(* PLC project mtcs_m3, Institute of Astronomy OntoManager 0.0.1 *)
(* stored: creationDateTime 2024-08-13T08:58:49.312185, modificationDateTime 2024-08-13T08:58:49.312185 *)

TYPE M3PositionIDs : (UNKNOWN := 0, CASSEGRAIN := 1, NASMYTH_A := 2, NASMYTH_B := 3, NASMYTH_C := 4, NASMYTH_D := 5, OTHER_0 := 6, OTHER_1 := 7, OTHER_2 := 8, OTHER_3 := 9, OTHER_4 := 10);
END_TYPE

TYPE M3GotoProcedureStates : (IDLE := 0, ABORTED := 1, PREPARE_PROCESS := 2, GOING_TO_POSITION := 3, IMPROVING_POSITION := 4, ERROR := 5, RESETTING := 6, ABORTING := 7);
END_TYPE

TYPE M3RotateProcedureStates : (IDLE := 0, ABORTED := 1, PREPARE_PROCESS := 2, DECOUPLING_AXES := 3, ENABLING_AXES := 4, UNDOING_OFFSET := 5, COUPLING_AXES := 6, BOTH_GOING_TO_TARGET_PLUS_OFFSET := 7, DECOUPLING_AXES_AGAIN := 8, MOVING_ABL_TO_FINAL_POSITION := 9, DISABLING_ABL := 10, MOVING_POS_TO_FINAL_POSITION := 11, IMPROVING_POSITION := 12, DISABLING_POS := 13, ERROR := 14, RESETTING := 15, ABORTING := 16);
END_TYPE

TYPE M3TranslateProcedureStates : (IDLE := 0, ABORTED := 1, PREPARE_PROCESS := 2, ENABLING_AXIS := 3, MOVING := 4, IMPROVING_POSITION := 5, DISABLING_AXIS := 6, ERROR := 7, RESETTING := 8, ABORTING := 9);
END_TYPE

TYPE M3TranslationHomingProcedureStates : (IDLE := 0, ABORTED := 1, PREPARE_PROCESS := 2, ENABLING_AXIS := 3, MOVE_TO_LIMIT_SWITCH := 4, WAIT_FOR_LIMIT_SWITCH := 5, STOP := 6, APPLY_HOMING_SETTINGS := 7, MOVE_TO_MECH_STOP := 8, WAIT_FOR_MECH_STOP := 9, SET_ZERO_POSITION := 10, DISABLE_AXIS := 11, RESETTING := 12, ERROR := 13, ABORTING := 14);
END_TYPE

TYPE M3CalibrateRotationProcedureStates : (IDLE := 0, ABORTED := 1, PREPARE_PROCESS := 2, DECOUPLING_AXES := 3, ENABLING_AXES := 4, COUPLING_AXES := 5, GOING_TO_START_POSITION := 6, DECOUPLING_AXES_AGAIN := 7, START_MOVING := 8, WAIT_UNTIL_MOVING_STABLE := 9, WAIT_UNTIL_RANGE_PASSED := 10, HALT := 11, GO_TO_CLUTCH_ZERO_TORQUE := 12, DISABLING_AXES := 13, WAIT_UNTIL_STANDSTILL := 14, SYNC_AXES := 15, ERROR := 16, RESETTING := 17, ABORTING := 18);
END_TYPE

TYPE M3TargetStates : (NO_TARGET_GIVEN := 0, KNOWN_POSITION := 1, NEW_POSITION := 2);
END_TYPE

TYPE M3Parts : STRUCT
  rotation : M3Rotation;  (* Rotation mechanism *)
  translation : M3Translation;  (* Translation mechanism *)
  io : M3IO;  (* I/O modules *)
  gotoProcedure : M3GotoProcedure;  (* The goto procedure *)
  configManager : ConfigManager;  (* The config manager (to load/save/activate configuration data) *)
END_STRUCT;
END_TYPE

TYPE M3RotationParts : STRUCT
  positioningAxis : AngularAxis;  (* Positioning axis: SSI encoder + Faulhaber drive *)
  antiBacklashAxis : AngularAxis;  (* Anti-backlash Axis: Faulhaber drive + hall sensors *)
  positioningDrive : FaulhaberDrive;  (* Positioning drive *)
  antiBacklashDrive : FaulhaberDrive;  (* Anti-backlash drive *)
  positioningHallAxis : AngularAxis;  (* Only hall sensors *)
  gotoProcedure : M3RotationGotoProcedure;  (* The goto procedure *)
  calibrateProcedure : M3RotationCalibrateProcedure;  (* The calibration procedure *)
END_STRUCT;
END_TYPE

TYPE M3TranslationParts : STRUCT
  motorAxis : LinearAxis;  (* Motor axis *)
  motorDrive : FaulhaberDrive;  (* Motor drive *)
  gotoProcedure : M3TranslationGotoProcedure;  (* The goto procedure *)
  homingProcedure : M3TranslationHomingProcedure;  (* The homing procedure *)
END_STRUCT;
END_TYPE

TYPE M3IOParts : STRUCT
  canOpenBus : CANopenBus;  (* CANopen bus *)
  coupler : EtherCatDevice;  (* Coupler *)
  slot1 : EtherCatDevice;  (* Slot 1 *)
  slot2 : EtherCatDevice;  (* Slot 2 *)
  slot3 : EtherCatDevice;  (* Slot 3 *)
  slot4 : EtherCatDevice;  (* Slot 4 *)
END_STRUCT;
END_TYPE

TYPE M3Processes : STRUCT
  initialize : Process;  (* Start initializing *)
  lock : Process;  (* Lock the system *)
  unlock : Process;  (* Unlock the system *)
  reset : Process;  (* Reset any errors *)
  changeOperatingState : ChangeOperatingStateProcess;  (* Change the operating state (e.g. AUTO, MANUAL, ...) *)
  gotoKnownPosition : M3GotoKnownPosition;  (* Go to the known position with the given name (only in AUTO mode!) *)
  gotoNewPosition : M3GotoNewPosition;  (* Go to the new position with the given settings (only in AUTO mode!) *)
  abort : Process;  (* Abort the goto procedure *)
END_STRUCT;
END_TYPE

TYPE M3RotationProcesses : STRUCT
  goto : M3RotationGoto;  (* Start moving the rotation stage to the given position *)
  abort : Process;  (* Abort any running procedures *)
  reset : Process;  (* Reset any errors *)
  calibrate : Process;  (* Start calibrating the rotation stage *)
END_STRUCT;
END_TYPE

TYPE M3TranslationProcesses : STRUCT
  goto : M3TranslationGoto;  (* Start moving the translation stage to the given position *)
  reset : Process;  (* Reset any errors *)
  abort : Process;  (* Abort any running procedures *)
  startHoming : Process;  (* Start the homing procedure *)
END_STRUCT;
END_TYPE

TYPE M3RotationTargetStatuses : STRUCT
  targetStatus : M3TargetStatus;
END_STRUCT;
END_TYPE

TYPE M3TranslationTargetStatuses : STRUCT
  targetStatus : M3TargetStatus;
END_STRUCT;
END_TYPE

TYPE M3Statuses : STRUCT
  initializationStatus : InitializationStatus;
  apertureStatus : ApertureStatus;
  healthStatus : HealthStatus;
  busyStatus : BusyStatus;
  operatingStatus : OperatingStatus;
END_STRUCT;
END_TYPE

TYPE M3GotoProcedureStatuses : STRUCT
  busyStatus : BusyStatus;  (* Is the M3GotoProcedure in a busy state? *)
  healthStatus : HealthStatus;  (* Is the M3GotoProcedure in a healthy state? *)
END_STRUCT;
END_TYPE

TYPE M3RotationStatuses : STRUCT
  healthStatus : HealthStatus;
  busyStatus : BusyStatus;
END_STRUCT;
END_TYPE

TYPE M3RotationGotoProcedureStatuses : STRUCT
  busyStatus : BusyStatus;  (* Is the M3RotationGotoProcedure in a busy state? *)
  healthStatus : HealthStatus;  (* Is the M3RotationGotoProcedure in a healthy state? *)
END_STRUCT;
END_TYPE

TYPE M3RotationCalibrateProcedureStatuses : STRUCT
  busyStatus : BusyStatus;  (* Is the M3RotationCalibrateProcedure in a busy state? *)
  healthStatus : HealthStatus;  (* Is the M3RotationCalibrateProcedure in a healthy state? *)
END_STRUCT;
END_TYPE

TYPE M3TranslationStatuses : STRUCT
  healthStatus : HealthStatus;
  busyStatus : BusyStatus;
END_STRUCT;
END_TYPE

TYPE M3TranslationGotoProcedureStatuses : STRUCT
  busyStatus : BusyStatus;  (* Is the M3GotoProcedure in a busy state? *)
  healthStatus : HealthStatus;  (* Is the M3GotoProcedure in a healthy state? *)
END_STRUCT;
END_TYPE

TYPE M3TranslationHomingProcedureStatuses : STRUCT
  busyStatus : BusyStatus;  (* Is the M3GotoProcedure in a busy state? *)
  healthStatus : HealthStatus;  (* Is the M3GotoProcedure in a healthy state? *)
END_STRUCT;
END_TYPE

TYPE M3IOStatuses : STRUCT
  healthStatus : HealthStatus;  (* Is the I/O in a healthy state? *)
END_STRUCT;
END_TYPE

TYPE M3PositionConfig : STRUCT
  name : STRING;  (* The name of the M3 position *)
  rotationPosition : LREAL;  (* The position of the rotation stage in degrees *)
  rotationOffset : LREAL;  (* The offset between the positions of the two motors of the rotation stage in degrees *)
  translationPosition : LREAL;  (* The position of the translation stage in millimeters *)
  doRotation : BOOL;  (* Do a rotation for this position (TRUE) or not (FALSE) *)
  doTranslation : BOOL;  (* Do a translation for this position (TRUE) or not (FALSE) *)
END_STRUCT;
END_TYPE

TYPE M3KnownPositionsConfig : STRUCT
  cassegrain : M3PositionConfig;  (* Cassegrain *)
  nasmythA : M3PositionConfig;  (* Nasmyth A *)
  nasmythB : M3PositionConfig;  (* Nasmyth B *)
  nasmythC : M3PositionConfig;  (* Nasmyth C *)
  nasmythD : M3PositionConfig;  (* Nasmyth D *)
  other0 : M3PositionConfig;  (* Freely choosable position 0 *)
  other1 : M3PositionConfig;  (* Freely choosable position 1 *)
  other2 : M3PositionConfig;  (* Freely choosable position 2 *)
  other3 : M3PositionConfig;  (* Freely choosable position 3 *)
  other4 : M3PositionConfig;  (* Freely choosable position 4 *)
END_STRUCT;
END_TYPE

TYPE M3RotationConfig : STRUCT
  standstillTolerance : LREAL;  (* The tolerance for which the axis appears to be standing still, in degrees/sec *)
  motorToMirrorRatio : LREAL;  (* The motor-to-mirror transmission ratio *)
  encoderToMirrorRatio : LREAL;  (* The encoder-to-mirror transmission ratio *)
  positioningDrive : FaulhaberDriveConfig;  (* The config of the positioning faulhaber drive *)
  antiBacklashDrive : FaulhaberDriveConfig;  (* The config of the anti-backlash faulhaber drive *)
  negativeSoftLimit : LREAL;  (* Negative soft limit, in degrees *)
  positiveSoftLimit : LREAL;  (* Negative soft limit, in degrees *)
  maxPositionError : LREAL;  (* Maximum position error, in degrees *)
  maxOffsetError : LREAL;  (* Maximum position error, in degrees *)
  gotoOffsetVelocity : LREAL;  (* Velocity to move from/to the offset position, in degrees/sec on the MOTOR reduction exit shaft reference system *)
  gotoTargetVelocity : LREAL;  (* Velocity to move to the target, in degrees/sec on the MIRROR reference system *)
  gotoImprovingPositionTime : LREAL;  (* Time while the Goto procedure may improve the position, in seconds *)
  calibrateStartPosition : LREAL;  (* Mirror position (in degrees) to start the calibration from *)
  calibrateMoveToZeroTorqueVelocity : LREAL;  (* Velocity to move to the zero-torque position, in degrees/sec on the MIRROR reference system *)
  calibrateVelocity : LREAL;  (* Velocity during which the current is being measured, in degrees/sec on the MIRROR reference system *)
  calibrateRange : LREAL;  (* Position range where the current is being measured, in degrees on the MOTOR reference system *)
  calibrateOffset : LREAL;  (* Degrees between zero-torque position and minimum-torque position, on the MOTOR reference system *)
END_STRUCT;
END_TYPE

TYPE M3TranslationConfig : STRUCT
  homingContinuousCurrentLimit : UINT;  (* The continuous current limit for the translation stage motor in milliAmps, during homing *)
  homingPeakCurrentLimit : UINT;  (* The peak current limit for the translation stage motor in milliAmps, during homing *)
  homingSearchLimitSwitchVelocity : LREAL;  (* The velocity of the motor shaft during homing, in mm/sec *)
  homingToHardwareStopVelocity : LREAL;  (* The velocity of the motor shaft during homing, in mm/sec *)
  standstillTolerance : LREAL;  (* The tolerance for which the axis appears to be standing still, in mm/sec *)
  motorDrive : FaulhaberDriveConfig;  (* The config of the faulhaber drive *)
  negativeSoftLimit : LREAL;  (* Negative soft limit, in millimeters *)
  positiveSoftLimit : LREAL;  (* Negative soft limit, in millimeters *)
  maxPositionError : LREAL;  (* Maximum position error, in millimeters *)
  drawCassegrainLimit : LREAL;  (* Below this limit (in millimeters) the mirror will be drawn flipped away *)
  drawNasmythLimit : LREAL;  (* Above this limit (in millimeters) the mirror will be drawn frontal *)
  gotoImprovingPositionTime : LREAL;  (* Time while the Goto procedure may improve the position, in seconds *)
  gotoVelocity : LREAL;  (* Velocity to go to a new position, in degrees/second *)
END_STRUCT;
END_TYPE

TYPE M3Config : STRUCT
  knownPositions : M3KnownPositionsConfig;  (* All known M3 positions *)
  rotation : M3RotationConfig;  (* The settings of the rotation stage *)
  translation : M3TranslationConfig;  (* The settings of the translation stage *)
  moveAfterInitialization : BOOL;  (* Move the mirror to a known position after initialization *)
  moveAfterInitializationPosition : STRING;  (* Move the mirror to this position after initialization *)
END_STRUCT;
END_TYPE

TYPE M3GotoKnownPositionArgs : STRUCT
  name : STRING;  (* Name of the position (must be configured in M3Config.knownPositions!) *)
END_STRUCT;
END_TYPE

TYPE M3GotoNewPositionArgs : STRUCT
  rotationPosition : LREAL;  (* Position of the rotation stage, in degrees *)
  rotationOffset : LREAL;  (* Offset between the motors of the rotation stage, in degrees *)
  translationPosition : LREAL;  (* Position of the rotation stage, in millimeters *)
  doRotation : BOOL;  (* Do a rotation for this position (TRUE) or not (FALSE) *)
  doTranslation : BOOL;  (* Do a translation for this position (TRUE) or not (FALSE) *)
END_STRUCT;
END_TYPE

TYPE M3RotationGotoArgs : STRUCT
  position : LREAL;  (* Position setpoint of the rotation stage, in degrees *)
  offset : LREAL;  (* Offset setpoint between the motors of the rotation stage, in degrees *)
END_STRUCT;
END_TYPE

TYPE M3TranslationGotoArgs : STRUCT
  position : LREAL;  (* Position setpoint of the translation stage, in millimeters *)
END_STRUCT;
END_TYPE

FUNCTION_BLOCK M3TargetStatus
  VAR_INPUT
    superState : BOOL := TRUE;  (* Super state (TRUE if the super state is active, or if there is no super state) *)
    state : M3TargetStates;  (* Enum! *)
  END_VAR
  VAR_OUTPUT
    {attribute 'OPC.UA.DA' := '1'}
    {attribute 'OPC.UA.DA.Access' := '1'}
    noTargetGiven : BOOL;  (* No target given *)
    {attribute 'OPC.UA.DA' := '1'}
    {attribute 'OPC.UA.DA.Access' := '1'}
    knownPosition : BOOL;  (* Known position *)
    {attribute 'OPC.UA.DA' := '1'}
    {attribute 'OPC.UA.DA.Access' := '1'}
    newPosition : BOOL;  (* Undefined *)
  END_VAR

            noTargetGiven := (state = M3TargetStates.NO_TARGET_GIVEN) AND superState;
knownPosition := (state = M3TargetStates.KNOWN_POSITION) AND superState;
newPosition := (state = M3TargetStates.NEW_POSITION) AND superState;

          
END_FUNCTION_BLOCK

FUNCTION_BLOCK SM_M3RotationTarget
  VAR_INPUT
    {attribute 'OPC.UA.DA' := '0'}
    isTargetGiven : BOOL;  (* TRUE if a target is given *)
    {attribute 'OPC.UA.DA' := '0'}
    newPositionDegrees : LREAL;  (* New target position in degrees *)
    {attribute 'OPC.UA.DA' := '0'}
    newOffsetDegrees : LREAL;  (* New target offset in degrees *)
  END_VAR
  VAR_OUTPUT
    {attribute 'OPC.UA.DA' := '1'}
    {attribute 'OPC.UA.DA.Access' := '1'}
    actualStatus : STRING;  (* Current status description *)
    previousStatus : STRING;  (* Previous status description *)
    {attribute 'OPC.UA.DA' := '1'}
    {attribute 'OPC.UA.DA.Access' := '1'}
    name : STRING;  (* Name of the target (only in case the position and offset match an entry in the config!) *)
    {attribute 'OPC.UA.DA' := '1'}
    {attribute 'OPC.UA.DA.Access' := '1'}
    position : AngularPosition;  (* Target position for M3 rotation (only in case statuses.targetStatus.noTargetGiven is FALSE) *)
    {attribute 'OPC.UA.DA' := '1'}
    {attribute 'OPC.UA.DA.Access' := '1'}
    offset : AngularPosition;  (* Target offset for M3 rotation (only in case statuses.targetStatus.noTargetGiven is FALSE) *)
    statuses : M3RotationTargetStatuses;  (* Statuses of the state machine *)
  END_VAR
  VAR_IN_OUT
    {attribute 'OPC.UA.DA' := '0'}
    knownPositions : M3KnownPositionsConfig;  (* The known positions *)
  END_VAR

            position( newDegreesValue := newPositionDegrees );
offset( newDegreesValue := newOffsetDegrees );
statuses.targetStatus();

          

{attribute 'TcRpcEnable' := '1'}
METHOD _log : BOOL
  VAR_INPUT
    name : STRING;  (* Name of this function block instance *)
  END_VAR
  VAR_IN_OUT
    buffer : LogBuffer;  (* Buffer to write all logging to *)
  END_VAR
  VAR
    subBuffer : LogBuffer;  (* Temporary buffer to write logging by parts (sub-statemachines) to *)
  END_VAR
                  LOGGER(
    name := name,
    actualStatus := THIS^.actualStatus,
    previousStatus := THIS^.previousStatus,
    buffer := buffer,
    subBuffer := subBuffer);

                
END_METHOD
END_FUNCTION_BLOCK

FUNCTION_BLOCK SM_M3TranslationTarget
  VAR_INPUT
    {attribute 'OPC.UA.DA' := '0'}
    isTargetGiven : BOOL := FALSE;  (* TRUE if a target is given *)
    {attribute 'OPC.UA.DA' := '0'}
    newPositionMillimeters : LREAL;  (* New target position in millimeters *)
  END_VAR
  VAR_OUTPUT
    {attribute 'OPC.UA.DA' := '1'}
    {attribute 'OPC.UA.DA.Access' := '1'}
    actualStatus : STRING;  (* Current status description *)
    previousStatus : STRING;  (* Previous status description *)
    {attribute 'OPC.UA.DA' := '1'}
    {attribute 'OPC.UA.DA.Access' := '1'}
    name : STRING;  (* Name of the target (only in case the position matches an entry in the config!) *)
    {attribute 'OPC.UA.DA' := '1'}
    {attribute 'OPC.UA.DA.Access' := '1'}
    position : LinearPosition;  (* Target position for M3 translation (only in case statuses.targetStatus.noTargetGiven is FALSE) *)
    statuses : M3TranslationTargetStatuses;  (* Statuses of the state machine *)
  END_VAR
  VAR_IN_OUT
    {attribute 'OPC.UA.DA' := '0'}
    knownPositions : M3KnownPositionsConfig;  (* The known positions *)
  END_VAR

            position( newMillimetersValue := newPositionMillimeters );
statuses.targetStatus();

          

{attribute 'TcRpcEnable' := '1'}
METHOD _log : BOOL
  VAR_INPUT
    name : STRING;  (* Name of this function block instance *)
  END_VAR
  VAR_IN_OUT
    buffer : LogBuffer;  (* Buffer to write all logging to *)
  END_VAR
  VAR
    subBuffer : LogBuffer;  (* Temporary buffer to write logging by parts (sub-statemachines) to *)
  END_VAR
                  LOGGER(
    name := name,
    actualStatus := THIS^.actualStatus,
    previousStatus := THIS^.previousStatus,
    buffer := buffer,
    subBuffer := subBuffer);

                
END_METHOD
END_FUNCTION_BLOCK

FUNCTION_BLOCK SM_M3
  VAR_INPUT
    {attribute 'OPC.UA.DA' := '1'}
    {attribute 'OPC.UA.DA.Access' := '1'}
    editableConfig : M3Config;  (* Editable configuration of M3 *)
  END_VAR
  VAR_OUTPUT
    {attribute 'OPC.UA.DA' := '1'}
    {attribute 'OPC.UA.DA.Access' := '1'}
    actualStatus : STRING;  (* Current status description *)
    previousStatus : STRING;  (* Previous status description *)
    {attribute 'OPC.UA.DA' := '1'}
    {attribute 'OPC.UA.DA.Access' := '1'}
    config : M3Config;  (* Active configuration of M3 *)
    {attribute 'OPC.UA.DA' := '1'}
    {attribute 'OPC.UA.DA.Access' := '1'}
    actualKnownPositionName : STRING;  (* Name of the actual position according to config.knownPositions *)
    {attribute 'OPC.UA.DA' := '1'}
    {attribute 'OPC.UA.DA.Access' := '1'}
    actualKnownPositionID : M3PositionIDs;  (* ID of the actual position according to config.knownPositions *)
    statuses : M3Statuses;  (* Statuses of the state machine *)
    parts : M3Parts;  (* Parts of the state machine *)
    processes : M3Processes;  (* Processes of the state machine *)
  END_VAR
  VAR_IN_OUT
    {attribute 'OPC.UA.DA' := '0'}
    operatorStatus : OperatorStatus;  (* Shared operator status *)
  END_VAR

            parts.rotation(
    initializationStatus := statuses.initializationStatus,
    operatorStatus := operatorStatus,
    operatingStatus := statuses.operatingStatus,
    config := config.rotation,
    m3Config := config);
parts.translation(
    initializationStatus := statuses.initializationStatus,
    operatorStatus := operatorStatus,
    operatingStatus := statuses.operatingStatus,
    config := config.translation,
    m3Config := config);
parts.io();
parts.gotoProcedure(
    rotation := parts.rotation,
    translation := parts.translation,
    m3Config := config);
parts.configManager( isEnabled := operatorStatus.tech );
statuses.initializationStatus();
statuses.apertureStatus();
statuses.healthStatus(
    isGood := parts.rotation.statuses.healthStatus.isGood AND (parts.translation.statuses.healthStatus.isGood AND (parts.gotoProcedure.statuses.healthStatus.isGood AND parts.io.statuses.healthStatus.isGood)),
    hasWarning := (parts.rotation.statuses.healthStatus.hasWarning OR (parts.translation.statuses.healthStatus.hasWarning OR (parts.gotoProcedure.statuses.healthStatus.hasWarning OR parts.io.statuses.healthStatus.hasWarning))) OR (statuses.busyStatus.idle AND (actualKnownPositionID = M3PositionIDs.UNKNOWN)));
statuses.busyStatus( isBusy := parts.rotation.statuses.busyStatus.busy OR (parts.translation.statuses.busyStatus.busy OR parts.gotoProcedure.statuses.busyStatus.busy) );
statuses.operatingStatus( superState := statuses.initializationStatus.initialized );
processes.initialize( isEnabled := statuses.initializationStatus.shutdown OR (statuses.initializationStatus.initializingFailed OR statuses.initializationStatus.initialized) );
processes.lock( isEnabled := operatorStatus.tech AND statuses.initializationStatus.initialized );
processes.unlock( isEnabled := operatorStatus.tech AND statuses.initializationStatus.locked );
processes.reset( isEnabled := statuses.healthStatus.bad );
processes.changeOperatingState( isEnabled := statuses.busyStatus.idle AND statuses.initializationStatus.initialized );
processes.gotoKnownPosition( isEnabled := parts.gotoProcedure.isGotoAllowed AND (statuses.initializationStatus.initialized AND statuses.operatingStatus.auto) );
processes.gotoNewPosition( isEnabled := parts.gotoProcedure.isGotoAllowed AND (statuses.initializationStatus.initialized AND statuses.operatingStatus.auto) );
processes.abort( isEnabled := parts.gotoProcedure.statuses.busyStatus.busy );

          

{attribute 'TcRpcEnable' := '1'}
METHOD initialize : RequestResults
                  initialize := THIS^.processes.initialize.request();

                
END_METHOD

{attribute 'TcRpcEnable' := '1'}
METHOD lock : RequestResults
                  lock := THIS^.processes.lock.request();

                
END_METHOD

{attribute 'TcRpcEnable' := '1'}
METHOD unlock : RequestResults
                  unlock := THIS^.processes.unlock.request();

                
END_METHOD

{attribute 'TcRpcEnable' := '1'}
METHOD reset : RequestResults
                  reset := THIS^.processes.reset.request();

                
END_METHOD

{attribute 'TcRpcEnable' := '1'}
METHOD changeOperatingState : RequestResults
  VAR_INPUT
    state : OperatingStates;
  END_VAR
                  changeOperatingState := THIS^.processes.changeOperatingState.request( state := state );

                
END_METHOD

{attribute 'TcRpcEnable' := '1'}
METHOD gotoKnownPosition : RequestResults
  VAR_INPUT
    name : STRING;
  END_VAR
                  gotoKnownPosition := THIS^.processes.gotoKnownPosition.request( name := name );

                
END_METHOD

{attribute 'TcRpcEnable' := '1'}
METHOD gotoNewPosition : RequestResults
  VAR_INPUT
    rotationPosition : LREAL;
    rotationOffset : LREAL;
    translationPosition : LREAL;
    doRotation : BOOL;
    doTranslation : BOOL;
  END_VAR
                  gotoNewPosition := THIS^.processes.gotoNewPosition.request(
    rotationPosition := rotationPosition,
    rotationOffset := rotationOffset,
    translationPosition := translationPosition,
    doRotation := doRotation,
    doTranslation := doTranslation);

                
END_METHOD

{attribute 'TcRpcEnable' := '1'}
METHOD abort : RequestResults
                  abort := THIS^.processes.abort.request();

                
END_METHOD

{attribute 'TcRpcEnable' := '1'}
METHOD _log : BOOL
  VAR_INPUT
    name : STRING;  (* Name of this function block instance *)
  END_VAR
  VAR_IN_OUT
    buffer : LogBuffer;  (* Buffer to write all logging to *)
  END_VAR
  VAR
    subBuffer : LogBuffer;  (* Temporary buffer to write logging by parts (sub-statemachines) to *)
  END_VAR
                  THIS^.parts.rotation._log(
    name := 'rotation',
    buffer := subBuffer);
THIS^.parts.translation._log(
    name := 'translation',
    buffer := subBuffer);
THIS^.parts.io._log(
    name := 'io',
    buffer := subBuffer);
THIS^.parts.gotoProcedure._log(
    name := 'gotoProcedure',
    buffer := subBuffer);
THIS^.parts.configManager._log(
    name := 'configManager',
    buffer := subBuffer);
THIS^.processes.initialize._log(
    name := 'processes.initialize',
    buffer := subBuffer);
THIS^.processes.lock._log(
    name := 'processes.lock',
    buffer := subBuffer);
THIS^.processes.unlock._log(
    name := 'processes.unlock',
    buffer := subBuffer);
THIS^.processes.reset._log(
    name := 'processes.reset',
    buffer := subBuffer);
THIS^.processes.changeOperatingState._log(
    name := 'processes.changeOperatingState',
    buffer := subBuffer);
THIS^.processes.gotoKnownPosition._log(
    name := 'processes.gotoKnownPosition',
    buffer := subBuffer);
THIS^.processes.gotoNewPosition._log(
    name := 'processes.gotoNewPosition',
    buffer := subBuffer);
THIS^.processes.abort._log(
    name := 'processes.abort',
    buffer := subBuffer);
LOGGER(
    name := name,
    actualStatus := THIS^.actualStatus,
    previousStatus := THIS^.previousStatus,
    buffer := buffer,
    subBuffer := subBuffer,
    pHealthStatus := ADR(THIS^.statuses.healthStatus),
    pBusyStatus := ADR(THIS^.statuses.busyStatus));

                
END_METHOD
END_FUNCTION_BLOCK

FUNCTION_BLOCK SM_M3GotoProcedure
  VAR_INPUT
    {attribute 'OPC.UA.DA' := '1'}
    {attribute 'OPC.UA.DA.Access' := '1'}
    state : M3GotoProcedureStates;  (* New state, to be set by the manual implementation *)
  END_VAR
  VAR_OUTPUT
    {attribute 'OPC.UA.DA' := '1'}
    {attribute 'OPC.UA.DA.Access' := '1'}
    actualStatus : STRING;  (* Current status description *)
    previousStatus : STRING;  (* Previous status description *)
    {attribute 'OPC.UA.DA' := '1'}
    {attribute 'OPC.UA.DA.Access' := '1'}
    isGotoAllowed : BOOL;  (* TRUE if a goto command is allowed *)
    statuses : M3GotoProcedureStatuses;  (* Statuses of the state machine *)
  END_VAR
  VAR_IN_OUT
    {attribute 'OPC.UA.DA' := '0'}
    rotation : M3Rotation;
    {attribute 'OPC.UA.DA' := '0'}
    translation : M3Translation;
    {attribute 'OPC.UA.DA' := '0'}
    m3Config : M3Config;
  END_VAR

            statuses.busyStatus( isBusy := NOT((state = M3GotoProcedureStates.IDLE) OR ((state = M3GotoProcedureStates.ABORTED) OR (state = M3GotoProcedureStates.ERROR))) );
statuses.healthStatus(
    isGood := NOT(state = M3GotoProcedureStates.ERROR),
    hasWarning := state = M3GotoProcedureStates.ABORTED);

          

{attribute 'TcRpcEnable' := '1'}
METHOD _log : BOOL
  VAR_INPUT
    name : STRING;  (* Name of this function block instance *)
  END_VAR
  VAR_IN_OUT
    buffer : LogBuffer;  (* Buffer to write all logging to *)
  END_VAR
  VAR
    subBuffer : LogBuffer;  (* Temporary buffer to write logging by parts (sub-statemachines) to *)
  END_VAR
                  LOGGER(
    name := name,
    actualStatus := THIS^.actualStatus,
    previousStatus := THIS^.previousStatus,
    buffer := buffer,
    subBuffer := subBuffer,
    pHealthStatus := ADR(THIS^.statuses.healthStatus),
    pBusyStatus := ADR(THIS^.statuses.busyStatus));

                
END_METHOD
END_FUNCTION_BLOCK

FUNCTION_BLOCK SM_M3Rotation
  VAR_INPUT
    {attribute 'OPC.UA.DA' := '1'}
    {attribute 'OPC.UA.DA.Access' := '1'}
    target : M3RotationTarget;
    {attribute 'OPC.UA.DA' := '1'}
    {attribute 'OPC.UA.DA.Access' := '1'}
    positiveLimitSwitchActive AT %I* : BOOL;  (* TRUE if the positive limit switch is active *)
    {attribute 'OPC.UA.DA' := '1'}
    {attribute 'OPC.UA.DA.Access' := '1'}
    negativeLimitSwitchActive AT %I* : BOOL;  (* TRUE if the negative limit switch is active *)
  END_VAR
  VAR_OUTPUT
    {attribute 'OPC.UA.DA' := '1'}
    {attribute 'OPC.UA.DA.Access' := '1'}
    actualStatus : STRING;  (* Current status description *)
    previousStatus : STRING;  (* Previous status description *)
    {attribute 'OPC.UA.DA' := '1'}
    {attribute 'OPC.UA.DA.Access' := '1'}
    actualPosition : AngularPosition;  (* The actual position of the rotation *)
    {attribute 'OPC.UA.DA' := '1'}
    {attribute 'OPC.UA.DA.Access' := '1'}
    actualPositionError : AngularPosition;  (* The actual position error of the rotation *)
    {attribute 'OPC.UA.DA' := '1'}
    {attribute 'OPC.UA.DA.Access' := '1'}
    actualOffset : AngularPosition;  (* The actual offset of the rotation *)
    {attribute 'OPC.UA.DA' := '1'}
    {attribute 'OPC.UA.DA.Access' := '1'}
    actualOffsetError : AngularPosition;  (* The actual offset error of the rotation *)
    statuses : M3RotationStatuses;  (* Statuses of the state machine *)
    parts : M3RotationParts;  (* Parts of the state machine *)
    processes : M3RotationProcesses;  (* Processes of the state machine *)
  END_VAR
  VAR_IN_OUT
    {attribute 'OPC.UA.DA' := '0'}
    initializationStatus : InitializationStatus;
    {attribute 'OPC.UA.DA' := '0'}
    operatorStatus : OperatorStatus;
    {attribute 'OPC.UA.DA' := '0'}
    operatingStatus : OperatingStatus;
    {attribute 'OPC.UA.DA' := '0'}
    config : M3RotationConfig;
    {attribute 'OPC.UA.DA' := '0'}
    m3Config : M3Config;
  END_VAR

            target( knownPositions := m3Config.knownPositions );
actualPosition( newDegreesValue := parts.positioningAxis.actPos.degrees.value );
actualPositionError( newDegreesValue := actualPosition.degrees.value - target.position.degrees.value );
actualOffset( newDegreesValue := parts.antiBacklashAxis.actPos.degrees.value - parts.positioningHallAxis.actPos.degrees.value );
actualOffsetError( newDegreesValue := actualOffset.degrees.value - target.offset.degrees.value );
parts.positioningAxis(
    isEnabled := operatorStatus.tech AND initializationStatus.initialized,
    standstillTolerance := config.standstillTolerance,
    isGearingSupported := FALSE);
parts.antiBacklashAxis(
    isEnabled := operatorStatus.tech AND initializationStatus.initialized,
    standstillTolerance := config.standstillTolerance * config.motorToMirrorRatio,
    isGearingSupported := TRUE);
parts.positioningDrive(
    isEnabled := operatorStatus.tech AND initializationStatus.initialized,
    config := config.positioningDrive);
parts.antiBacklashDrive(
    isEnabled := operatorStatus.tech AND initializationStatus.initialized,
    config := config.antiBacklashDrive);
parts.positioningHallAxis(
    isEnabled := FALSE,
    standstillTolerance := config.standstillTolerance * config.motorToMirrorRatio,
    isGearingSupported := FALSE);
parts.gotoProcedure(
    config := config,
    positioningAxis := parts.positioningAxis,
    antiBacklashAxis := parts.antiBacklashAxis,
    positioningDrive := parts.positioningDrive,
    antiBacklashDrive := parts.antiBacklashDrive,
    positioningHallAxis := parts.positioningHallAxis,
    target := target,
    positiveLimitSwitchActive := positiveLimitSwitchActive,
    negativeLimitSwitchActive := negativeLimitSwitchActive,
    actualPosition := actualPosition,
    actualPositionError := actualPositionError,
    actualOffset := actualOffset,
    actualOffsetError := actualOffsetError);
parts.calibrateProcedure(
    config := config,
    positioningAxis := parts.positioningAxis,
    antiBacklashAxis := parts.antiBacklashAxis,
    positioningDrive := parts.positioningDrive,
    antiBacklashDrive := parts.antiBacklashDrive,
    positioningHallAxis := parts.positioningHallAxis,
    target := target,
    actualPosition := actualPosition,
    actualPositionError := actualPositionError,
    actualOffset := actualOffset,
    actualOffsetError := actualOffsetError);
statuses.healthStatus(
    isGood := parts.positioningAxis.statuses.healthStatus.isGood AND (parts.antiBacklashAxis.statuses.healthStatus.isGood AND (parts.positioningDrive.statuses.healthStatus.isGood AND (parts.antiBacklashDrive.statuses.healthStatus.isGood AND (parts.positioningHallAxis.statuses.healthStatus.isGood AND parts.gotoProcedure.statuses.healthStatus.isGood)))),
    hasWarning := parts.positioningAxis.statuses.healthStatus.hasWarning OR (parts.antiBacklashAxis.statuses.healthStatus.hasWarning OR (parts.positioningDrive.statuses.healthStatus.hasWarning OR (parts.antiBacklashDrive.statuses.healthStatus.hasWarning OR (parts.positioningHallAxis.statuses.healthStatus.hasWarning OR parts.gotoProcedure.statuses.healthStatus.hasWarning)))));
statuses.busyStatus( isBusy := parts.positioningAxis.statuses.busyStatus.busy OR (parts.antiBacklashAxis.statuses.busyStatus.busy OR (parts.positioningDrive.statuses.busyStatus.busy OR (parts.antiBacklashDrive.statuses.busyStatus.busy OR parts.gotoProcedure.statuses.busyStatus.busy))) );
processes.goto( isEnabled := operatingStatus.manual AND (initializationStatus.initialized AND parts.gotoProcedure.isGotoAllowed) );
processes.abort( isEnabled := parts.gotoProcedure.statuses.busyStatus.busy OR parts.calibrateProcedure.statuses.busyStatus.busy );
processes.reset( isEnabled := statuses.healthStatus.bad );
processes.calibrate( isEnabled := operatingStatus.manual AND initializationStatus.initialized );

          

{attribute 'TcRpcEnable' := '1'}
METHOD goto : RequestResults
  VAR_INPUT
    position : LREAL;
    offset : LREAL;
  END_VAR
                  goto := THIS^.processes.goto.request(
    position := position,
    offset := offset);

                
END_METHOD

{attribute 'TcRpcEnable' := '1'}
METHOD abort : RequestResults
                  abort := THIS^.processes.abort.request();

                
END_METHOD

{attribute 'TcRpcEnable' := '1'}
METHOD reset : RequestResults
                  reset := THIS^.processes.reset.request();

                
END_METHOD

{attribute 'TcRpcEnable' := '1'}
METHOD calibrate : RequestResults
                  calibrate := THIS^.processes.calibrate.request();

                
END_METHOD

{attribute 'TcRpcEnable' := '1'}
METHOD _log : BOOL
  VAR_INPUT
    name : STRING;  (* Name of this function block instance *)
  END_VAR
  VAR_IN_OUT
    buffer : LogBuffer;  (* Buffer to write all logging to *)
  END_VAR
  VAR
    subBuffer : LogBuffer;  (* Temporary buffer to write logging by parts (sub-statemachines) to *)
  END_VAR
                  THIS^.parts.positioningAxis._log(
    name := 'positioningAxis',
    buffer := subBuffer);
THIS^.parts.antiBacklashAxis._log(
    name := 'antiBacklashAxis',
    buffer := subBuffer);
THIS^.parts.positioningDrive._log(
    name := 'positioningDrive',
    buffer := subBuffer);
THIS^.parts.antiBacklashDrive._log(
    name := 'antiBacklashDrive',
    buffer := subBuffer);
THIS^.parts.positioningHallAxis._log(
    name := 'positioningHallAxis',
    buffer := subBuffer);
THIS^.parts.gotoProcedure._log(
    name := 'gotoProcedure',
    buffer := subBuffer);
THIS^.parts.calibrateProcedure._log(
    name := 'calibrateProcedure',
    buffer := subBuffer);
THIS^.processes.goto._log(
    name := 'processes.goto',
    buffer := subBuffer);
THIS^.processes.abort._log(
    name := 'processes.abort',
    buffer := subBuffer);
THIS^.processes.reset._log(
    name := 'processes.reset',
    buffer := subBuffer);
THIS^.processes.calibrate._log(
    name := 'processes.calibrate',
    buffer := subBuffer);
LOGGER(
    name := name,
    actualStatus := THIS^.actualStatus,
    previousStatus := THIS^.previousStatus,
    buffer := buffer,
    subBuffer := subBuffer,
    pHealthStatus := ADR(THIS^.statuses.healthStatus),
    pBusyStatus := ADR(THIS^.statuses.busyStatus));

                
END_METHOD
END_FUNCTION_BLOCK

FUNCTION_BLOCK SM_M3RotationGotoProcedure
  VAR_INPUT
    {attribute 'OPC.UA.DA' := '1'}
    {attribute 'OPC.UA.DA.Access' := '1'}
    state : M3RotateProcedureStates;  (* New state, to be set by the manual implementation *)
  END_VAR
  VAR_OUTPUT
    {attribute 'OPC.UA.DA' := '1'}
    {attribute 'OPC.UA.DA.Access' := '1'}
    actualStatus : STRING;  (* Current status description *)
    previousStatus : STRING;  (* Previous status description *)
    {attribute 'OPC.UA.DA' := '1'}
    {attribute 'OPC.UA.DA.Access' := '1'}
    isGotoAllowed : BOOL;  (* TRUE if a goto command is allowed *)
    statuses : M3RotationGotoProcedureStatuses;  (* Statuses of the state machine *)
  END_VAR
  VAR_IN_OUT
    {attribute 'OPC.UA.DA' := '0'}
    config : M3RotationConfig;
    {attribute 'OPC.UA.DA' := '0'}
    positioningAxis : AngularAxis;
    {attribute 'OPC.UA.DA' := '0'}
    antiBacklashAxis : AngularAxis;
    {attribute 'OPC.UA.DA' := '0'}
    positioningDrive : FaulhaberDrive;
    {attribute 'OPC.UA.DA' := '0'}
    antiBacklashDrive : FaulhaberDrive;
    {attribute 'OPC.UA.DA' := '0'}
    positioningHallAxis : AngularAxis;
    {attribute 'OPC.UA.DA' := '0'}
    target : M3RotationTarget;
    {attribute 'OPC.UA.DA' := '0'}
    positiveLimitSwitchActive : BOOL;
    {attribute 'OPC.UA.DA' := '0'}
    negativeLimitSwitchActive : BOOL;
    {attribute 'OPC.UA.DA' := '0'}
    actualPosition : AngularPosition;
    {attribute 'OPC.UA.DA' := '0'}
    actualPositionError : AngularPosition;
    {attribute 'OPC.UA.DA' := '0'}
    actualOffset : AngularPosition;
    {attribute 'OPC.UA.DA' := '0'}
    actualOffsetError : AngularPosition;
  END_VAR

            statuses.busyStatus( isBusy := NOT((state = M3RotateProcedureStates.IDLE) OR ((state = M3RotateProcedureStates.ABORTED) OR (state = M3RotateProcedureStates.ERROR))) );
statuses.healthStatus(
    isGood := NOT(state = M3RotateProcedureStates.ERROR),
    hasWarning := state = M3RotateProcedureStates.ABORTED);

          

{attribute 'TcRpcEnable' := '1'}
METHOD _log : BOOL
  VAR_INPUT
    name : STRING;  (* Name of this function block instance *)
  END_VAR
  VAR_IN_OUT
    buffer : LogBuffer;  (* Buffer to write all logging to *)
  END_VAR
  VAR
    subBuffer : LogBuffer;  (* Temporary buffer to write logging by parts (sub-statemachines) to *)
  END_VAR
                  LOGGER(
    name := name,
    actualStatus := THIS^.actualStatus,
    previousStatus := THIS^.previousStatus,
    buffer := buffer,
    subBuffer := subBuffer,
    pHealthStatus := ADR(THIS^.statuses.healthStatus),
    pBusyStatus := ADR(THIS^.statuses.busyStatus));

                
END_METHOD
END_FUNCTION_BLOCK

FUNCTION_BLOCK SM_M3RotationCalibrateProcedure
  VAR_INPUT
    {attribute 'OPC.UA.DA' := '1'}
    {attribute 'OPC.UA.DA.Access' := '1'}
    state : M3CalibrateRotationProcedureStates;  (* Current state of the *)
  END_VAR
  VAR_OUTPUT
    {attribute 'OPC.UA.DA' := '1'}
    {attribute 'OPC.UA.DA.Access' := '1'}
    actualStatus : STRING;  (* Current status description *)
    previousStatus : STRING;  (* Previous status description *)
    statuses : M3RotationCalibrateProcedureStatuses;  (* Statuses of the state machine *)
  END_VAR
  VAR_IN_OUT
    {attribute 'OPC.UA.DA' := '0'}
    config : M3RotationConfig;
    {attribute 'OPC.UA.DA' := '0'}
    positioningAxis : AngularAxis;
    {attribute 'OPC.UA.DA' := '0'}
    antiBacklashAxis : AngularAxis;
    {attribute 'OPC.UA.DA' := '0'}
    positioningDrive : FaulhaberDrive;
    {attribute 'OPC.UA.DA' := '0'}
    antiBacklashDrive : FaulhaberDrive;
    {attribute 'OPC.UA.DA' := '0'}
    positioningHallAxis : AngularAxis;
    {attribute 'OPC.UA.DA' := '0'}
    target : M3RotationTarget;
    {attribute 'OPC.UA.DA' := '0'}
    actualPosition : AngularPosition;
    {attribute 'OPC.UA.DA' := '0'}
    actualPositionError : AngularPosition;
    {attribute 'OPC.UA.DA' := '0'}
    actualOffset : AngularPosition;
    {attribute 'OPC.UA.DA' := '0'}
    actualOffsetError : AngularPosition;
  END_VAR

            statuses.busyStatus( isBusy := NOT((state = M3CalibrateRotationProcedureStates.IDLE) OR ((state = M3CalibrateRotationProcedureStates.ABORTED) OR (state = M3CalibrateRotationProcedureStates.ERROR))) );
statuses.healthStatus(
    isGood := NOT(state = M3CalibrateRotationProcedureStates.ERROR),
    hasWarning := state = M3CalibrateRotationProcedureStates.ABORTED);

          

{attribute 'TcRpcEnable' := '1'}
METHOD _log : BOOL
  VAR_INPUT
    name : STRING;  (* Name of this function block instance *)
  END_VAR
  VAR_IN_OUT
    buffer : LogBuffer;  (* Buffer to write all logging to *)
  END_VAR
  VAR
    subBuffer : LogBuffer;  (* Temporary buffer to write logging by parts (sub-statemachines) to *)
  END_VAR
                  LOGGER(
    name := name,
    actualStatus := THIS^.actualStatus,
    previousStatus := THIS^.previousStatus,
    buffer := buffer,
    subBuffer := subBuffer,
    pHealthStatus := ADR(THIS^.statuses.healthStatus),
    pBusyStatus := ADR(THIS^.statuses.busyStatus));

                
END_METHOD
END_FUNCTION_BLOCK

FUNCTION_BLOCK SM_M3Translation
  VAR_INPUT
    {attribute 'OPC.UA.DA' := '1'}
    {attribute 'OPC.UA.DA.Access' := '1'}
    target : M3TranslationTarget;
    {attribute 'OPC.UA.DA' := '1'}
    {attribute 'OPC.UA.DA.Access' := '1'}
    positiveLimitSwitchActive AT %I* : BOOL;  (* TRUE if the positive limit switch is active *)
    {attribute 'OPC.UA.DA' := '1'}
    {attribute 'OPC.UA.DA.Access' := '1'}
    negativeLimitSwitchActive AT %I* : BOOL;  (* TRUE if the negative limit switch is active *)
  END_VAR
  VAR_OUTPUT
    {attribute 'OPC.UA.DA' := '1'}
    {attribute 'OPC.UA.DA.Access' := '1'}
    actualStatus : STRING;  (* Current status description *)
    previousStatus : STRING;  (* Previous status description *)
    {attribute 'OPC.UA.DA' := '1'}
    {attribute 'OPC.UA.DA.Access' := '1'}
    actualPosition : LinearPosition;  (* The actual position of the translation *)
    {attribute 'OPC.UA.DA' := '1'}
    {attribute 'OPC.UA.DA.Access' := '1'}
    actualPositionError : LinearPosition;  (* The actual position error of the translation *)
    statuses : M3TranslationStatuses;  (* Statuses of the state machine *)
    parts : M3TranslationParts;  (* Parts of the state machine *)
    processes : M3TranslationProcesses;  (* Processes of the state machine *)
  END_VAR
  VAR_IN_OUT
    {attribute 'OPC.UA.DA' := '0'}
    initializationStatus : InitializationStatus;
    {attribute 'OPC.UA.DA' := '0'}
    operatorStatus : OperatorStatus;
    {attribute 'OPC.UA.DA' := '0'}
    operatingStatus : OperatingStatus;
    {attribute 'OPC.UA.DA' := '0'}
    config : M3TranslationConfig;
    {attribute 'OPC.UA.DA' := '0'}
    m3Config : M3Config;
  END_VAR

            target( knownPositions := m3Config.knownPositions );
actualPosition( newMillimetersValue := parts.motorAxis.actPos.millimeters.value );
actualPositionError( newMillimetersValue := actualPosition.millimeters.value - target.position.millimeters.value );
parts.motorAxis(
    isEnabled := operatorStatus.tech AND initializationStatus.initialized,
    standstillTolerance := config.standstillTolerance,
    isGearingSupported := FALSE);
parts.motorDrive(
    isEnabled := operatorStatus.tech AND initializationStatus.initialized,
    config := config.motorDrive);
parts.gotoProcedure(
    config := config,
    motorAxis := parts.motorAxis,
    motorDrive := parts.motorDrive,
    target := target,
    positiveLimitSwitchActive := positiveLimitSwitchActive,
    negativeLimitSwitchActive := negativeLimitSwitchActive,
    actualPosition := actualPosition,
    actualPositionError := actualPositionError);
parts.homingProcedure(
    config := config,
    motorAxis := parts.motorAxis,
    motorDrive := parts.motorDrive,
    target := target,
    positiveLimitSwitchActive := positiveLimitSwitchActive,
    negativeLimitSwitchActive := negativeLimitSwitchActive,
    actualPosition := actualPosition,
    actualPositionError := actualPositionError);
statuses.healthStatus(
    isGood := parts.motorAxis.statuses.healthStatus.isGood AND (parts.motorDrive.statuses.healthStatus.isGood AND (parts.homingProcedure.statuses.healthStatus.isGood AND parts.gotoProcedure.statuses.healthStatus.isGood)),
    hasWarning := parts.motorAxis.statuses.healthStatus.hasWarning OR (parts.motorDrive.statuses.healthStatus.hasWarning OR (parts.homingProcedure.statuses.healthStatus.hasWarning OR parts.gotoProcedure.statuses.healthStatus.hasWarning)));
statuses.busyStatus( isBusy := parts.motorAxis.statuses.busyStatus.busy );
processes.goto( isEnabled := operatingStatus.manual AND (initializationStatus.initialized AND parts.gotoProcedure.isGotoAllowed) );
processes.reset( isEnabled := statuses.healthStatus.bad );
processes.abort( isEnabled := parts.gotoProcedure.statuses.busyStatus.busy OR parts.homingProcedure.statuses.busyStatus.busy );
processes.startHoming( isEnabled := operatingStatus.manual AND initializationStatus.initialized );

          

{attribute 'TcRpcEnable' := '1'}
METHOD goto : RequestResults
  VAR_INPUT
    position : LREAL;
  END_VAR
                  goto := THIS^.processes.goto.request( position := position );

                
END_METHOD

{attribute 'TcRpcEnable' := '1'}
METHOD reset : RequestResults
                  reset := THIS^.processes.reset.request();

                
END_METHOD

{attribute 'TcRpcEnable' := '1'}
METHOD abort : RequestResults
                  abort := THIS^.processes.abort.request();

                
END_METHOD

{attribute 'TcRpcEnable' := '1'}
METHOD startHoming : RequestResults
                  startHoming := THIS^.processes.startHoming.request();

                
END_METHOD

{attribute 'TcRpcEnable' := '1'}
METHOD _log : BOOL
  VAR_INPUT
    name : STRING;  (* Name of this function block instance *)
  END_VAR
  VAR_IN_OUT
    buffer : LogBuffer;  (* Buffer to write all logging to *)
  END_VAR
  VAR
    subBuffer : LogBuffer;  (* Temporary buffer to write logging by parts (sub-statemachines) to *)
  END_VAR
                  THIS^.parts.motorAxis._log(
    name := 'motorAxis',
    buffer := subBuffer);
THIS^.parts.motorDrive._log(
    name := 'motorDrive',
    buffer := subBuffer);
THIS^.parts.gotoProcedure._log(
    name := 'gotoProcedure',
    buffer := subBuffer);
THIS^.parts.homingProcedure._log(
    name := 'homingProcedure',
    buffer := subBuffer);
THIS^.processes.goto._log(
    name := 'processes.goto',
    buffer := subBuffer);
THIS^.processes.reset._log(
    name := 'processes.reset',
    buffer := subBuffer);
THIS^.processes.abort._log(
    name := 'processes.abort',
    buffer := subBuffer);
THIS^.processes.startHoming._log(
    name := 'processes.startHoming',
    buffer := subBuffer);
LOGGER(
    name := name,
    actualStatus := THIS^.actualStatus,
    previousStatus := THIS^.previousStatus,
    buffer := buffer,
    subBuffer := subBuffer,
    pHealthStatus := ADR(THIS^.statuses.healthStatus),
    pBusyStatus := ADR(THIS^.statuses.busyStatus));

                
END_METHOD
END_FUNCTION_BLOCK

FUNCTION_BLOCK SM_M3TranslationGotoProcedure
  VAR_INPUT
    {attribute 'OPC.UA.DA' := '1'}
    {attribute 'OPC.UA.DA.Access' := '1'}
    state : M3TranslateProcedureStates;  (* New state, to be set by the manual implementation *)
  END_VAR
  VAR_OUTPUT
    {attribute 'OPC.UA.DA' := '1'}
    {attribute 'OPC.UA.DA.Access' := '1'}
    actualStatus : STRING;  (* Current status description *)
    previousStatus : STRING;  (* Previous status description *)
    {attribute 'OPC.UA.DA' := '1'}
    {attribute 'OPC.UA.DA.Access' := '1'}
    isGotoAllowed : BOOL;  (* TRUE if a goto command is allowed *)
    statuses : M3TranslationGotoProcedureStatuses;  (* Statuses of the state machine *)
  END_VAR
  VAR_IN_OUT
    {attribute 'OPC.UA.DA' := '0'}
    config : M3TranslationConfig;
    {attribute 'OPC.UA.DA' := '0'}
    motorAxis : LinearAxis;
    {attribute 'OPC.UA.DA' := '0'}
    motorDrive : FaulhaberDrive;
    {attribute 'OPC.UA.DA' := '0'}
    target : M3TranslationTarget;
    {attribute 'OPC.UA.DA' := '0'}
    positiveLimitSwitchActive : BOOL;
    {attribute 'OPC.UA.DA' := '0'}
    negativeLimitSwitchActive : BOOL;
    {attribute 'OPC.UA.DA' := '0'}
    actualPosition : LinearPosition;
    {attribute 'OPC.UA.DA' := '0'}
    actualPositionError : LinearPosition;
  END_VAR

            statuses.busyStatus( isBusy := NOT((state = M3TranslateProcedureStates.IDLE) OR ((state = M3TranslateProcedureStates.ABORTED) OR (state = M3TranslateProcedureStates.ERROR))) );
statuses.healthStatus(
    isGood := NOT(state = M3TranslateProcedureStates.ERROR),
    hasWarning := state = M3TranslateProcedureStates.ABORTED);

          

{attribute 'TcRpcEnable' := '1'}
METHOD _log : BOOL
  VAR_INPUT
    name : STRING;  (* Name of this function block instance *)
  END_VAR
  VAR_IN_OUT
    buffer : LogBuffer;  (* Buffer to write all logging to *)
  END_VAR
  VAR
    subBuffer : LogBuffer;  (* Temporary buffer to write logging by parts (sub-statemachines) to *)
  END_VAR
                  LOGGER(
    name := name,
    actualStatus := THIS^.actualStatus,
    previousStatus := THIS^.previousStatus,
    buffer := buffer,
    subBuffer := subBuffer,
    pHealthStatus := ADR(THIS^.statuses.healthStatus),
    pBusyStatus := ADR(THIS^.statuses.busyStatus));

                
END_METHOD
END_FUNCTION_BLOCK

FUNCTION_BLOCK SM_M3TranslationHomingProcedure
  VAR_INPUT
    {attribute 'OPC.UA.DA' := '1'}
    {attribute 'OPC.UA.DA.Access' := '1'}
    state : M3TranslationHomingProcedureStates;  (* State to be set by the manual implementation *)
  END_VAR
  VAR_OUTPUT
    {attribute 'OPC.UA.DA' := '1'}
    {attribute 'OPC.UA.DA.Access' := '1'}
    actualStatus : STRING;  (* Current status description *)
    previousStatus : STRING;  (* Previous status description *)
    statuses : M3TranslationHomingProcedureStatuses;  (* Statuses of the state machine *)
  END_VAR
  VAR_IN_OUT
    {attribute 'OPC.UA.DA' := '0'}
    config : M3TranslationConfig;
    {attribute 'OPC.UA.DA' := '0'}
    motorAxis : LinearAxis;
    {attribute 'OPC.UA.DA' := '0'}
    motorDrive : FaulhaberDrive;
    {attribute 'OPC.UA.DA' := '0'}
    target : M3TranslationTarget;
    {attribute 'OPC.UA.DA' := '0'}
    positiveLimitSwitchActive : BOOL;
    {attribute 'OPC.UA.DA' := '0'}
    negativeLimitSwitchActive : BOOL;
    {attribute 'OPC.UA.DA' := '0'}
    actualPosition : LinearPosition;
    {attribute 'OPC.UA.DA' := '0'}
    actualPositionError : LinearPosition;
  END_VAR

            statuses.busyStatus( isBusy := NOT((state = M3TranslationHomingProcedureStates.IDLE) OR ((state = M3TranslationHomingProcedureStates.ABORTED) OR (state = M3TranslationHomingProcedureStates.ERROR))) );
statuses.healthStatus(
    isGood := NOT(state = M3TranslationHomingProcedureStates.ERROR),
    hasWarning := state = M3TranslationHomingProcedureStates.ABORTED);

          

{attribute 'TcRpcEnable' := '1'}
METHOD _log : BOOL
  VAR_INPUT
    name : STRING;  (* Name of this function block instance *)
  END_VAR
  VAR_IN_OUT
    buffer : LogBuffer;  (* Buffer to write all logging to *)
  END_VAR
  VAR
    subBuffer : LogBuffer;  (* Temporary buffer to write logging by parts (sub-statemachines) to *)
  END_VAR
                  LOGGER(
    name := name,
    actualStatus := THIS^.actualStatus,
    previousStatus := THIS^.previousStatus,
    buffer := buffer,
    subBuffer := subBuffer,
    pHealthStatus := ADR(THIS^.statuses.healthStatus),
    pBusyStatus := ADR(THIS^.statuses.busyStatus));

                
END_METHOD
END_FUNCTION_BLOCK

FUNCTION_BLOCK SM_M3IO
  VAR_OUTPUT
    {attribute 'OPC.UA.DA' := '1'}
    {attribute 'OPC.UA.DA.Access' := '1'}
    actualStatus : STRING;  (* Current status description *)
    previousStatus : STRING;  (* Previous status description *)
    statuses : M3IOStatuses;  (* Statuses of the state machine *)
    parts : M3IOParts;  (* Parts of the state machine *)
  END_VAR

            parts.canOpenBus();
parts.coupler(
    id := 'COUPLER',
    typeId := 'EK1101');
parts.slot1(
    id := 'IODI1',
    typeId := 'EL1088');
parts.slot2(
    id := 'IOEN1',
    typeId := 'EL5101');
parts.slot3(
    id := 'IOEN2',
    typeId := 'EL5001');
parts.slot4(
    id := 'IOCO1',
    typeId := 'EL6751');
statuses.healthStatus(
    isGood := parts.coupler.statuses.healthStatus.isGood AND (parts.slot1.statuses.healthStatus.isGood AND (parts.slot2.statuses.healthStatus.isGood AND (parts.slot3.statuses.healthStatus.isGood AND parts.slot4.statuses.healthStatus.isGood))),
    hasWarning := parts.coupler.statuses.healthStatus.hasWarning OR (parts.slot1.statuses.healthStatus.hasWarning OR (parts.slot2.statuses.healthStatus.hasWarning OR (parts.slot3.statuses.healthStatus.hasWarning OR parts.slot4.statuses.healthStatus.hasWarning))));

          

{attribute 'TcRpcEnable' := '1'}
METHOD _log : BOOL
  VAR_INPUT
    name : STRING;  (* Name of this function block instance *)
  END_VAR
  VAR_IN_OUT
    buffer : LogBuffer;  (* Buffer to write all logging to *)
  END_VAR
  VAR
    subBuffer : LogBuffer;  (* Temporary buffer to write logging by parts (sub-statemachines) to *)
  END_VAR
                  THIS^.parts.canOpenBus._log(
    name := 'canOpenBus',
    buffer := subBuffer);
THIS^.parts.coupler._log(
    name := 'coupler',
    buffer := subBuffer);
THIS^.parts.slot1._log(
    name := 'slot1',
    buffer := subBuffer);
THIS^.parts.slot2._log(
    name := 'slot2',
    buffer := subBuffer);
THIS^.parts.slot3._log(
    name := 'slot3',
    buffer := subBuffer);
THIS^.parts.slot4._log(
    name := 'slot4',
    buffer := subBuffer);
LOGGER(
    name := name,
    actualStatus := THIS^.actualStatus,
    previousStatus := THIS^.previousStatus,
    buffer := buffer,
    subBuffer := subBuffer,
    pHealthStatus := ADR(THIS^.statuses.healthStatus));

                
END_METHOD
END_FUNCTION_BLOCK

FUNCTION_BLOCK M3GotoKnownPosition EXTENDS BaseProcess
  VAR_INPUT
    {attribute 'OPC.UA.DA' := '1'}
    set : M3GotoKnownPositionArgs;  (* Arguments to be set, before writing do_request TRUE *)
  END_VAR
  VAR_OUTPUT
    {attribute 'OPC.UA.DA' := '1'}
    {attribute 'OPC.UA.DA.Access' := '1'}
    get : M3GotoKnownPositionArgs;  (* Arguments in use by the process, if do_request was accepted *)
  END_VAR

            IF do_request THEN
    do_request_result := request( name := set.name );
    do_request := FALSE;
END_IF;
SUPER^();

          

{attribute 'TcRpcEnable' := '1'}
METHOD start
  VAR_INPUT
    name : STRING;  (* Name of the position (must be configured in M3Config.knownPositions!) *)
  END_VAR
                  THIS^.get.name := name;
THIS^.statuses.busyStatus( isBusy := TRUE );
THIS^.statuses.healthStatus( isGood := TRUE );

                
END_METHOD

{attribute 'TcRpcEnable' := '1'}
METHOD request : RequestResults
  VAR_INPUT
    name : STRING;  (* Name of the position (must be configured in M3Config.knownPositions!) *)
  END_VAR
                  IF THIS^.statuses.enabledStatus.enabled THEN
    request := RequestResults.ACCEPTED;
    THIS^.start( name := name );
ELSE
    request := RequestResults.REJECTED;
END_IF;

                
END_METHOD
END_FUNCTION_BLOCK

FUNCTION_BLOCK M3GotoNewPosition EXTENDS BaseProcess
  VAR_INPUT
    {attribute 'OPC.UA.DA' := '1'}
    set : M3GotoNewPositionArgs;  (* Arguments to be set, before writing do_request TRUE *)
  END_VAR
  VAR_OUTPUT
    {attribute 'OPC.UA.DA' := '1'}
    {attribute 'OPC.UA.DA.Access' := '1'}
    get : M3GotoNewPositionArgs;  (* Arguments in use by the process, if do_request was accepted *)
  END_VAR

            IF do_request THEN
    do_request_result := request(
    rotationPosition := set.rotationPosition,
    rotationOffset := set.rotationOffset,
    translationPosition := set.translationPosition,
    doRotation := set.doRotation,
    doTranslation := set.doTranslation);
    do_request := FALSE;
END_IF;
SUPER^();

          

{attribute 'TcRpcEnable' := '1'}
METHOD start
  VAR_INPUT
    rotationPosition : LREAL;  (* Position of the rotation stage, in degrees *)
    rotationOffset : LREAL;  (* Offset between the motors of the rotation stage, in degrees *)
    translationPosition : LREAL;  (* Position of the rotation stage, in millimeters *)
    doRotation : BOOL;  (* Do a rotation for this position (TRUE) or not (FALSE) *)
    doTranslation : BOOL;  (* Do a translation for this position (TRUE) or not (FALSE) *)
  END_VAR
                  THIS^.get.rotationPosition := rotationPosition;
THIS^.get.rotationOffset := rotationOffset;
THIS^.get.translationPosition := translationPosition;
THIS^.get.doRotation := doRotation;
THIS^.get.doTranslation := doTranslation;
THIS^.statuses.busyStatus( isBusy := TRUE );
THIS^.statuses.healthStatus( isGood := TRUE );

                
END_METHOD

{attribute 'TcRpcEnable' := '1'}
METHOD request : RequestResults
  VAR_INPUT
    rotationPosition : LREAL;  (* Position of the rotation stage, in degrees *)
    rotationOffset : LREAL;  (* Offset between the motors of the rotation stage, in degrees *)
    translationPosition : LREAL;  (* Position of the rotation stage, in millimeters *)
    doRotation : BOOL;  (* Do a rotation for this position (TRUE) or not (FALSE) *)
    doTranslation : BOOL;  (* Do a translation for this position (TRUE) or not (FALSE) *)
  END_VAR
                  IF THIS^.statuses.enabledStatus.enabled THEN
    request := RequestResults.ACCEPTED;
    THIS^.start(
        rotationPosition := rotationPosition,
        rotationOffset := rotationOffset,
        translationPosition := translationPosition,
        doRotation := doRotation,
        doTranslation := doTranslation);
ELSE
    request := RequestResults.REJECTED;
END_IF;

                
END_METHOD
END_FUNCTION_BLOCK

FUNCTION_BLOCK M3RotationGoto EXTENDS BaseProcess
  VAR_INPUT
    {attribute 'OPC.UA.DA' := '1'}
    set : M3RotationGotoArgs;  (* Arguments to be set, before writing do_request TRUE *)
  END_VAR
  VAR_OUTPUT
    {attribute 'OPC.UA.DA' := '1'}
    {attribute 'OPC.UA.DA.Access' := '1'}
    get : M3RotationGotoArgs;  (* Arguments in use by the process, if do_request was accepted *)
  END_VAR

            IF do_request THEN
    do_request_result := request(
    position := set.position,
    offset := set.offset);
    do_request := FALSE;
END_IF;
SUPER^();

          

{attribute 'TcRpcEnable' := '1'}
METHOD start
  VAR_INPUT
    position : LREAL;  (* Position setpoint of the rotation stage, in degrees *)
    offset : LREAL;  (* Offset setpoint between the motors of the rotation stage, in degrees *)
  END_VAR
                  THIS^.get.position := position;
THIS^.get.offset := offset;
THIS^.statuses.busyStatus( isBusy := TRUE );
THIS^.statuses.healthStatus( isGood := TRUE );

                
END_METHOD

{attribute 'TcRpcEnable' := '1'}
METHOD request : RequestResults
  VAR_INPUT
    position : LREAL;  (* Position setpoint of the rotation stage, in degrees *)
    offset : LREAL;  (* Offset setpoint between the motors of the rotation stage, in degrees *)
  END_VAR
                  IF THIS^.statuses.enabledStatus.enabled THEN
    request := RequestResults.ACCEPTED;
    THIS^.start(
        position := position,
        offset := offset);
ELSE
    request := RequestResults.REJECTED;
END_IF;

                
END_METHOD
END_FUNCTION_BLOCK

FUNCTION_BLOCK M3TranslationGoto EXTENDS BaseProcess
  VAR_INPUT
    {attribute 'OPC.UA.DA' := '1'}
    set : M3TranslationGotoArgs;  (* Arguments to be set, before writing do_request TRUE *)
  END_VAR
  VAR_OUTPUT
    {attribute 'OPC.UA.DA' := '1'}
    {attribute 'OPC.UA.DA.Access' := '1'}
    get : M3TranslationGotoArgs;  (* Arguments in use by the process, if do_request was accepted *)
  END_VAR

            IF do_request THEN
    do_request_result := request( position := set.position );
    do_request := FALSE;
END_IF;
SUPER^();

          

{attribute 'TcRpcEnable' := '1'}
METHOD start
  VAR_INPUT
    position : LREAL;  (* Position setpoint of the translation stage, in millimeters *)
  END_VAR
                  THIS^.get.position := position;
THIS^.statuses.busyStatus( isBusy := TRUE );
THIS^.statuses.healthStatus( isGood := TRUE );

                
END_METHOD

{attribute 'TcRpcEnable' := '1'}
METHOD request : RequestResults
  VAR_INPUT
    position : LREAL;  (* Position setpoint of the translation stage, in millimeters *)
  END_VAR
                  IF THIS^.statuses.enabledStatus.enabled THEN
    request := RequestResults.ACCEPTED;
    THIS^.start( position := position );
ELSE
    request := RequestResults.REJECTED;
END_IF;

                
END_METHOD
END_FUNCTION_BLOCK
